PROGRAM ProgramTask1
VAR
	fbSpscBuff 	: FB_SpscBuffer;
	ipSpscBuff 	: I_SpscBuffer 		:= fbSpscBuff;
	nCounter 	: UDINT;
	bInit 		: BOOL;
END_VAR

nCounter := nCounter + 1;
IF NOT(binit) THEN
	bInit := TRUE;
	ipSpscBuff.Initialize(SIZEOF(UDINT),100);
END_IF

ipSpscBuff.Push(ADR(nCounter),SIZEOF(nCounter));
ipSpscBuff.Reset();

END_PROGRAM

(* stored: Version 1.1.0.1
   POU ProgramTask1: Id {e90d93f6-babc-4924-ad7f-966aed5b6722}, SpecialFunc None *)
